Omron CX-Programmer project NewProject (CX-Programmer 9.73)

# PLC tombol_cerdas_cermat: CJ2M CPU11

## Global symbols (name address type ; comment)
tombol_siram 0.00 BOOL  ; Tombol siram manual
tombol_auto 0.01 BOOL  ; Tombol toggle mode otomatis
pompa 100.00 BOOL  ; Output pompa penyiraman
mode_auto H0.00 BOOL  ; Flag mode otomatis aktif
trigger_siram W0.00 BOOL  ; Trigger siram aktif
oneshot_1 W0.03 BOOL  ; One-shot jadwal 1
oneshot_2 W0.04 BOOL  ; One-shot jadwal 2
timer_siram T0 BOOL  ; Timer durasi siram
jam_rtc W10 WORD  ; Jam BCD dari RTC
menit_rtc W11 WORD  ; Menit BCD dari RTC
jam_1 D0 WORD  ; Jam jadwal 1 default=6
menit_1 D1 WORD  ; Menit jadwal 1 default=0
jam_2 D2 WORD  ; Jam jadwal 2 default=16
menit_2 D3 WORD  ; Menit jadwal 2 default=0
durasi_siram D4 WORD  ; Durasi siram x100ms default=300
tombol_pupuk 0.02 BOOL  ; Tombol pupuk manual
pupuk 101.00 BOOL  ; Output solenoid pupuk
tombol_lampu_on 0.03 BOOL  ; Tombol lampu ON manual
tombol_lampu_off 0.04 BOOL  ; Tombol lampu OFF manual
lampu 102.00 BOOL  ; Output lampu
flag_lampu_manual H0.01 BOOL  ; Flag lampu ON manual latch
flag_lampu_auto H0.02 BOOL  ; Flag lampu ON otomatis
flag_lampu_override H0.03 BOOL  ; Flag override paksa OFF lampu
tombol_emergency 0.05 BOOL  ; Tombol emergency reset semua
jam_lampu_on D10 WORD  ; Jam nyala lampu default=18
jam_lampu_off D11 WORD  ; Jam mati lampu default=6

## Program NewProgram1 (cyclic task 0)

### Section Penyiraman

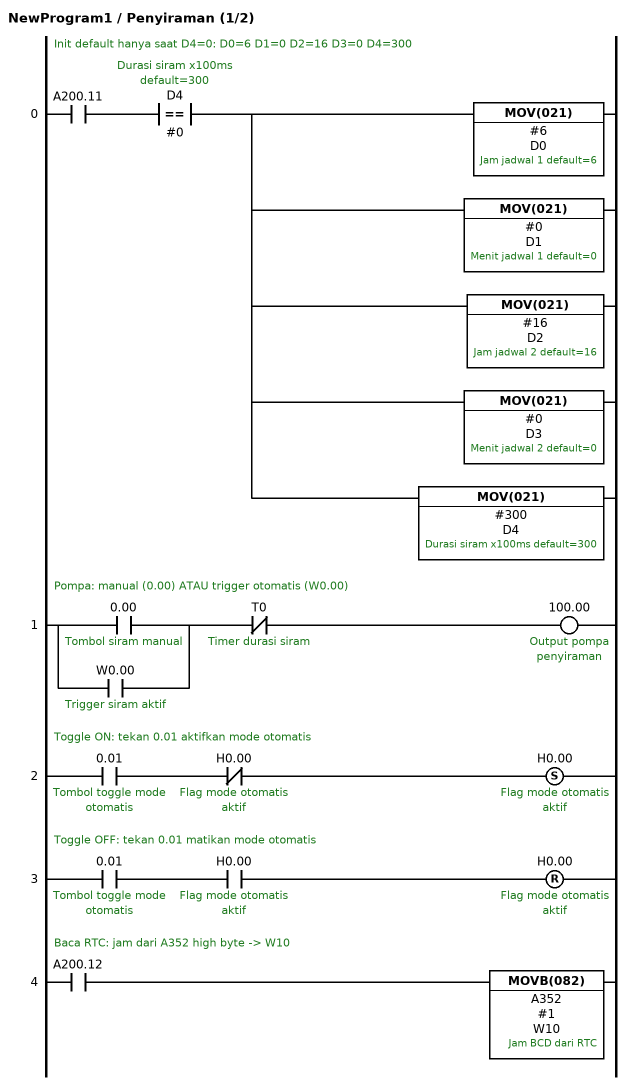
; rung 0: Init default hanya saat D4=0: D0=6 D1=0 D2=16 D3=0 D4=300
LD A200.11
AND= D4 #0  ; Durasi siram x100ms default=300
MOV(021) #6 D0  ; Jam jadwal 1 default=6
MOV(021) #0 D1  ; Menit jadwal 1 default=0
MOV(021) #16 D2  ; Jam jadwal 2 default=16
MOV(021) #0 D3  ; Menit jadwal 2 default=0
MOV(021) #300 D4  ; Durasi siram x100ms default=300
; rung 1: Pompa: manual (0.00) ATAU trigger otomatis (W0.00)
LD 0.00  ; Tombol siram manual
OR W0.00  ; Trigger siram aktif
ANDNOT T0  ; Timer durasi siram
OUT 100.00  ; Output pompa penyiraman
; rung 2: Toggle ON: tekan 0.01 aktifkan mode otomatis
LD 0.01  ; Tombol toggle mode otomatis
ANDNOT H0.00  ; Flag mode otomatis aktif
SET H0.00  ; Flag mode otomatis aktif
; rung 3: Toggle OFF: tekan 0.01 matikan mode otomatis
LD 0.01  ; Tombol toggle mode otomatis
AND H0.00  ; Flag mode otomatis aktif
RSET H0.00  ; Flag mode otomatis aktif
; rung 4: Baca RTC: jam dari A352 high byte -> W10
LD A200.12
MOVB(082) A352 #1 W10  ; Jam BCD dari RTC

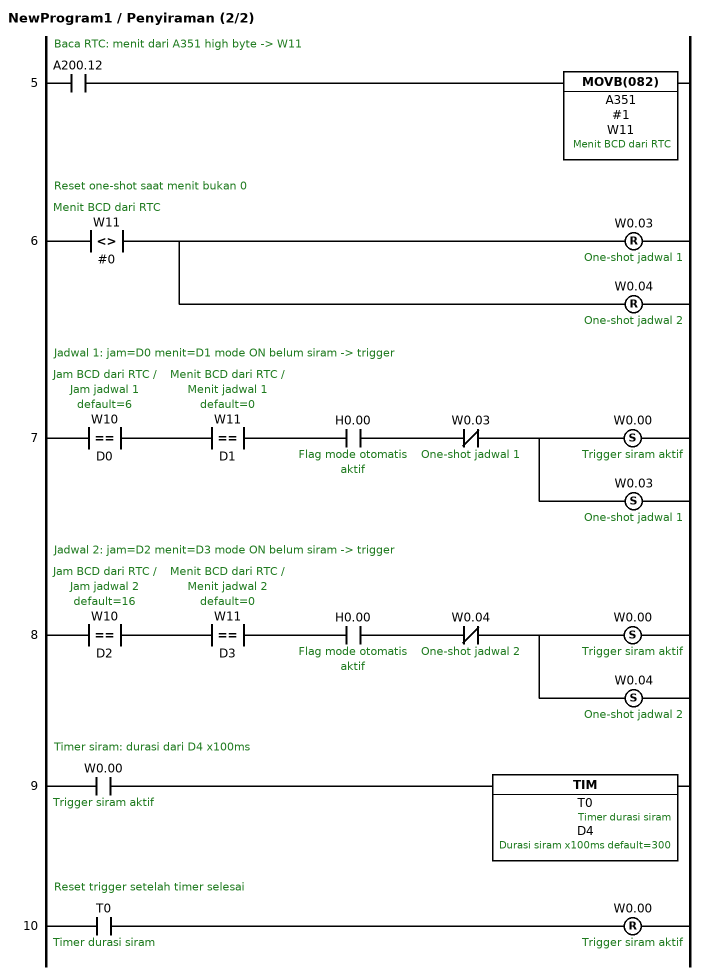
; rung 5: Baca RTC: menit dari A351 high byte -> W11
LD A200.12
MOVB(082) A351 #1 W11  ; Menit BCD dari RTC
; rung 6: Reset one-shot saat menit bukan 0
LD<> W11 #0  ; Menit BCD dari RTC
RSET W0.03  ; One-shot jadwal 1
RSET W0.04  ; One-shot jadwal 2
; rung 7: Jadwal 1: jam=D0 menit=D1 mode ON belum siram -> trigger
LD= W10 D0  ; Jam BCD dari RTC, Jam jadwal 1 default=6
AND= W11 D1  ; Menit BCD dari RTC, Menit jadwal 1 default=0
AND H0.00  ; Flag mode otomatis aktif
ANDNOT W0.03  ; One-shot jadwal 1
SET W0.00  ; Trigger siram aktif
SET W0.03  ; One-shot jadwal 1
; rung 8: Jadwal 2: jam=D2 menit=D3 mode ON belum siram -> trigger
LD= W10 D2  ; Jam BCD dari RTC, Jam jadwal 2 default=16
AND= W11 D3  ; Menit BCD dari RTC, Menit jadwal 2 default=0
AND H0.00  ; Flag mode otomatis aktif
ANDNOT W0.04  ; One-shot jadwal 2
SET W0.00  ; Trigger siram aktif
SET W0.04  ; One-shot jadwal 2
; rung 9: Timer siram: durasi dari D4 x100ms
LD W0.00  ; Trigger siram aktif
TIM T0 D4  ; Timer durasi siram, Durasi siram x100ms default=300
; rung 10: Reset trigger setelah timer selesai
LD T0  ; Timer durasi siram
RSET W0.00  ; Trigger siram aktif

### Section Pupuk

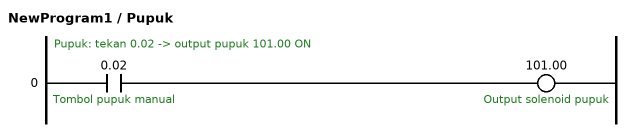
; rung 0: Pupuk: tekan 0.02 -> output pupuk 101.00 ON
LD 0.02  ; Tombol pupuk manual
OUT 101.00  ; Output solenoid pupuk

### Section Lampu

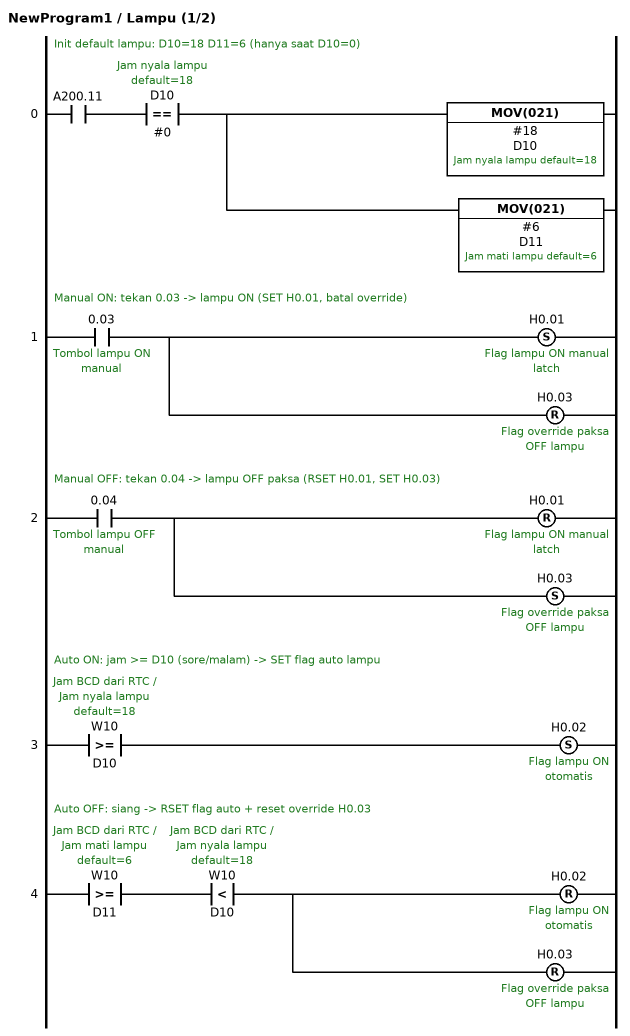
; rung 0: Init default lampu: D10=18 D11=6 (hanya saat D10=0)
LD A200.11
AND= D10 #0  ; Jam nyala lampu default=18
MOV(021) #18 D10  ; Jam nyala lampu default=18
MOV(021) #6 D11  ; Jam mati lampu default=6
; rung 1: Manual ON: tekan 0.03 -> lampu ON (SET H0.01, batal override)
LD 0.03  ; Tombol lampu ON manual
SET H0.01  ; Flag lampu ON manual latch
RSET H0.03  ; Flag override paksa OFF lampu
; rung 2: Manual OFF: tekan 0.04 -> lampu OFF paksa (RSET H0.01, SET H0.03)
LD 0.04  ; Tombol lampu OFF manual
RSET H0.01  ; Flag lampu ON manual latch
SET H0.03  ; Flag override paksa OFF lampu
; rung 3: Auto ON: jam >= D10 (sore/malam) -> SET flag auto lampu
LD>= W10 D10  ; Jam BCD dari RTC, Jam nyala lampu default=18
SET H0.02  ; Flag lampu ON otomatis
; rung 4: Auto OFF: siang -> RSET flag auto + reset override H0.03
LD>= W10 D11  ; Jam BCD dari RTC, Jam mati lampu default=6
AND< W10 D10  ; Jam BCD dari RTC, Jam nyala lampu default=18
RSET H0.02  ; Flag lampu ON otomatis
RSET H0.03  ; Flag override paksa OFF lampu

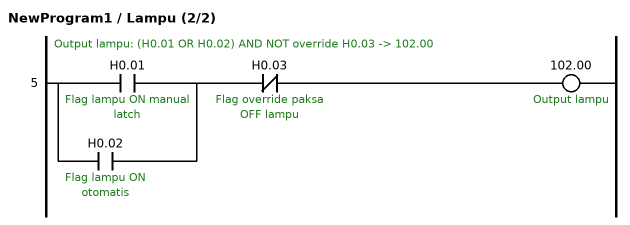
; rung 5: Output lampu: (H0.01 OR H0.02) AND NOT override H0.03 -> 102.00
LD H0.01  ; Flag lampu ON manual latch
OR H0.02  ; Flag lampu ON otomatis
ANDNOT H0.03  ; Flag override paksa OFF lampu
OUT 102.00  ; Output lampu

### Section Emergency

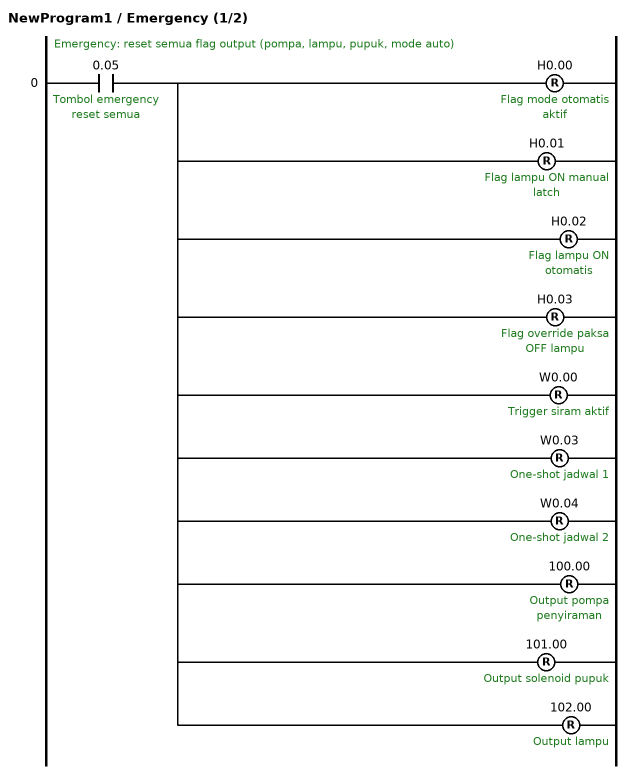
; rung 0: Emergency: reset semua flag output (pompa, lampu, pupuk, mode auto)
LD 0.05  ; Tombol emergency reset semua
RSET H0.00  ; Flag mode otomatis aktif
RSET H0.01  ; Flag lampu ON manual latch
RSET H0.02  ; Flag lampu ON otomatis
RSET H0.03  ; Flag override paksa OFF lampu
RSET W0.00  ; Trigger siram aktif
RSET W0.03  ; One-shot jadwal 1
RSET W0.04  ; One-shot jadwal 2
RSET 100.00  ; Output pompa penyiraman
RSET 101.00  ; Output solenoid pupuk
RSET 102.00  ; Output lampu

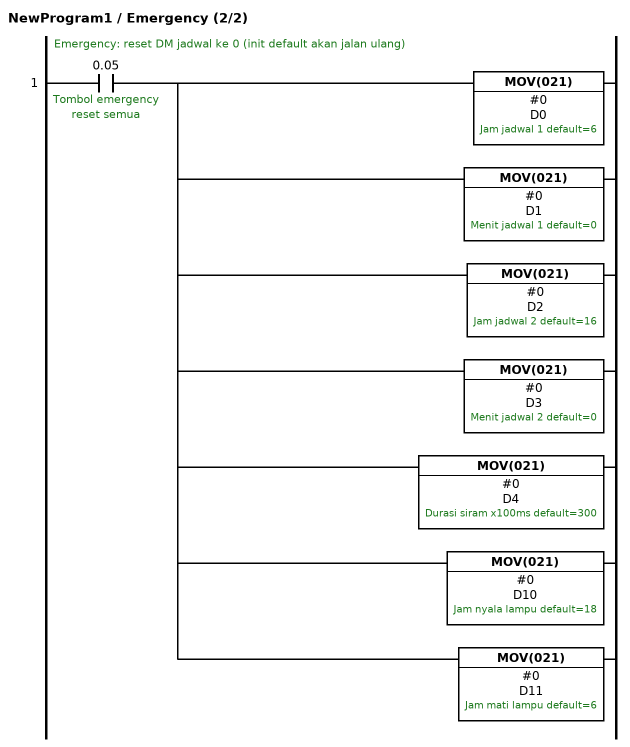
; rung 1: Emergency: reset DM jadwal ke 0 (init default akan jalan ulang)
LD 0.05  ; Tombol emergency reset semua
MOV(021) #0 D0  ; Jam jadwal 1 default=6
MOV(021) #0 D1  ; Menit jadwal 1 default=0
MOV(021) #0 D2  ; Jam jadwal 2 default=16
MOV(021) #0 D3  ; Menit jadwal 2 default=0
MOV(021) #0 D4  ; Durasi siram x100ms default=300
MOV(021) #0 D10  ; Jam nyala lampu default=18
MOV(021) #0 D11  ; Jam mati lampu default=6

### Section END
; rung 0
END(001)